# EPICS substitutions: apps/mpodLvApp/Db/bonus-hv.substitutions
file "db/mpod-crate.db" {
    pattern { HOST }
    { hvbonus2 }
}

file "db/iseg-module.db" {
    pattern {HOST HOSTNAME MX}
    {129.57.86.181 hvbonus2 1 }
    {129.57.86.181 hvbonus2 2 }
}

file "db/iseg-channel.db" {
    pattern {HVHOST HV HVCH}
    { 129.57.86.181 B_BONUS_HV_GEM3_OUT 1  }
    { 129.57.86.181 B_BONUS_HV_GEM3_IN  2  }
    { 129.57.86.181 B_BONUS_HV_GEM2_OUT 3  }
    { 129.57.86.181 B_BONUS_HV_GEM2_IN  4  }
    { 129.57.86.181 B_BONUS_HV_GEM1_OUT 5  }
    { 129.57.86.181 B_BONUS_HV_GEM1_IN  6  }
    { 129.57.86.181 B_BONUS_HV_CATHODE 101 }
}

file "db/caenhv_genericStat.db" {
    pattern {P}
    {B_BONUS_HV}
}
